// TIA Portal V19 export
FUNCTION_BLOCK "F_TwoHands_FB"   // FB93, F_LAD
TITLE = SAFE BUTTONS - TWO HANDS / ENABLING SWITCH / DEAD-MAN
// stored: Access Published
   VAR
      LB101 : "TwoHand_FB";
      LB111 : "TwoHand_FB";
      LB112 : "TwoHand_FB";
      LB113 : "TwoHand_FB";
      LB113_Welder : "TwoHand_FB";
      LB114_FeedA01 : "TwoHand_FB";
      LB114_FeedA02 : "TwoHand_FB";
      LB131 : "TwoHand_FB";
      LB131_FeedA01 : "TwoHand_FB";
      LB211 : "TwoHand_FB";
      LB212_FlyC : "TwoHand_FB";
      LB212_FeedA03 : "TwoHand_FB";
      LB311 : "TwoHand_FB";
   END_VAR
BEGIN

REGION Network 1: <<<< AREA 01 >>>
END_REGION

REGION Network 2: LB101 Two hands @ Zone 01 (Front of decoiler in load) / LB1.1 Two hands @ Area 01 Zone 01 (Front of decoiler in load)
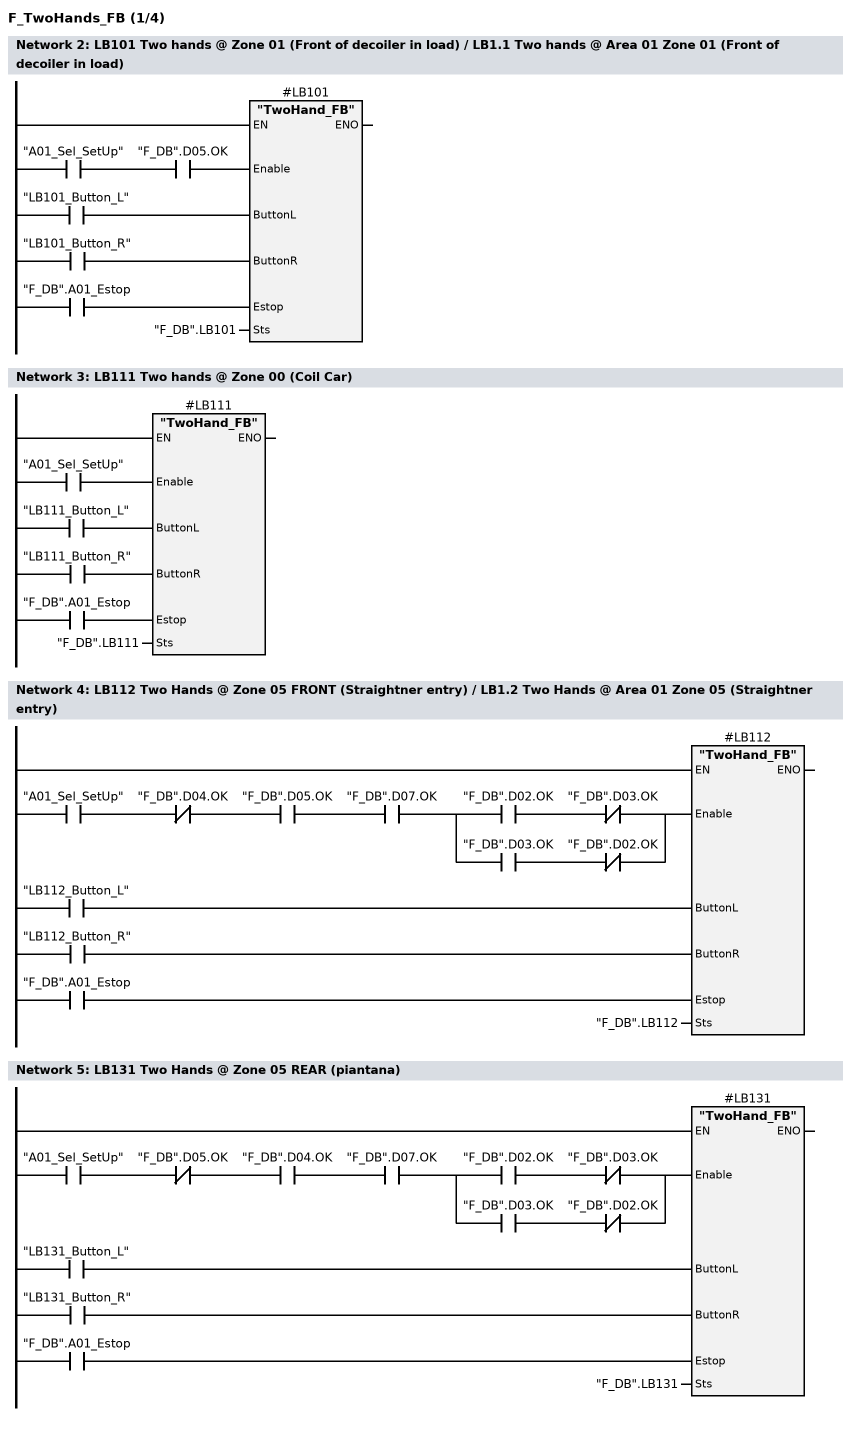
   RUNG wire#powerrail
      #LB101(Enable := wire#w1, ButtonL := wire#w2, ButtonR := wire#w3, Estop := wire#w4, Sts := "F_DB".LB101)
   END_RUNG
   RUNG wire#powerrail
      Contact( "A01_Sel_SetUp" )
      Contact( "F_DB".D05.OK )
   END_RUNG wire#w1
   RUNG wire#powerrail
      Contact( "LB101_Button_L" )
   END_RUNG wire#w2
   RUNG wire#powerrail
      Contact( "LB101_Button_R" )
   END_RUNG wire#w3
   RUNG wire#powerrail
      Contact( "F_DB".A01_Estop )
   END_RUNG wire#w4
   // the same network as SCL:
   #LB101(Enable := "A01_Sel_SetUp" AND "F_DB".D05.OK,   // "TwoHand_FB"
          ButtonL := "LB101_Button_L",
          ButtonR := "LB101_Button_R",
          Estop := "F_DB".A01_Estop,
          Sts := "F_DB".LB101);
END_REGION

REGION Network 3: LB111 Two hands @ Zone 00 (Coil Car)
   RUNG wire#powerrail
      #LB111(Enable := wire#w1, ButtonL := wire#w2, ButtonR := wire#w3, Estop := wire#w4, Sts := "F_DB".LB111)
   END_RUNG
   RUNG wire#powerrail
      Contact( "A01_Sel_SetUp" )
   END_RUNG wire#w1
   RUNG wire#powerrail
      Contact( "LB111_Button_L" )
   END_RUNG wire#w2
   RUNG wire#powerrail
      Contact( "LB111_Button_R" )
   END_RUNG wire#w3
   RUNG wire#powerrail
      Contact( "F_DB".A01_Estop )
   END_RUNG wire#w4
   // the same network as SCL:
   #LB111(Enable := "A01_Sel_SetUp",   // "TwoHand_FB"
          ButtonL := "LB111_Button_L",
          ButtonR := "LB111_Button_R",
          Estop := "F_DB".A01_Estop,
          Sts := "F_DB".LB111);
END_REGION

REGION Network 4: LB112 Two Hands @ Zone 05 FRONT (Straightner entry) / LB1.2 Two Hands @ Area 01 Zone 05 (Straightner entry)
   RUNG wire#powerrail
      #LB112(Enable := wire#w2, ButtonL := wire#w3, ButtonR := wire#w4, Estop := wire#w5, Sts := "F_DB".LB112)
   END_RUNG
   RUNG wire#powerrail
      Contact( "A01_Sel_SetUp" )
      I_Contact( "F_DB".D04.OK )
      Contact( "F_DB".D05.OK )
      Contact( "F_DB".D07.OK )
      wire#w1
      Contact( "F_DB".D02.OK )
      I_Contact( "F_DB".D03.OK )
   END_RUNG wire#w2
   RUNG wire#w1
      Contact( "F_DB".D03.OK )
      I_Contact( "F_DB".D02.OK )
   END_RUNG wire#w2
   RUNG wire#powerrail
      Contact( "LB112_Button_L" )
   END_RUNG wire#w3
   RUNG wire#powerrail
      Contact( "LB112_Button_R" )
   END_RUNG wire#w4
   RUNG wire#powerrail
      Contact( "F_DB".A01_Estop )
   END_RUNG wire#w5
   // the same network as SCL:
   #LB112(Enable := "A01_Sel_SetUp" AND NOT "F_DB".D04.OK AND "F_DB".D05.OK AND "F_DB".D07.OK AND (("F_DB".D02.OK AND NOT "F_DB".D03.OK) OR ("F_DB".D03.OK AND NOT "F_DB".D02.OK)),   // "TwoHand_FB"
          ButtonL := "LB112_Button_L",
          ButtonR := "LB112_Button_R",
          Estop := "F_DB".A01_Estop,
          Sts := "F_DB".LB112);
END_REGION

REGION Network 5: LB131 Two Hands @ Zone 05 REAR (piantana)
   RUNG wire#powerrail
      #LB131(Enable := wire#w2, ButtonL := wire#w3, ButtonR := wire#w4, Estop := wire#w5, Sts := "F_DB".LB131)
   END_RUNG
   RUNG wire#powerrail
      Contact( "A01_Sel_SetUp" )
      I_Contact( "F_DB".D05.OK )
      Contact( "F_DB".D04.OK )
      Contact( "F_DB".D07.OK )
      wire#w1
      Contact( "F_DB".D02.OK )
      I_Contact( "F_DB".D03.OK )
   END_RUNG wire#w2
   RUNG wire#w1
      Contact( "F_DB".D03.OK )
      I_Contact( "F_DB".D02.OK )
   END_RUNG wire#w2
   RUNG wire#powerrail
      Contact( "LB131_Button_L" )
   END_RUNG wire#w3
   RUNG wire#powerrail
      Contact( "LB131_Button_R" )
   END_RUNG wire#w4
   RUNG wire#powerrail
      Contact( "F_DB".A01_Estop )
   END_RUNG wire#w5
   // the same network as SCL:
   #LB131(Enable := "A01_Sel_SetUp" AND NOT "F_DB".D05.OK AND "F_DB".D04.OK AND "F_DB".D07.OK AND (("F_DB".D02.OK AND NOT "F_DB".D03.OK) OR ("F_DB".D03.OK AND NOT "F_DB".D02.OK)),   // "TwoHand_FB"
          ButtonL := "LB131_Button_L",
          ButtonR := "LB131_Button_R",
          Estop := "F_DB".A01_Estop,
          Sts := "F_DB".LB131);
END_REGION

REGION Network 6: LB113 Two Hands @ Zone 05 FRONT (Junction bench) / LB1.3 Two Hands @ Area 01 Zone 07 (Junction bench)
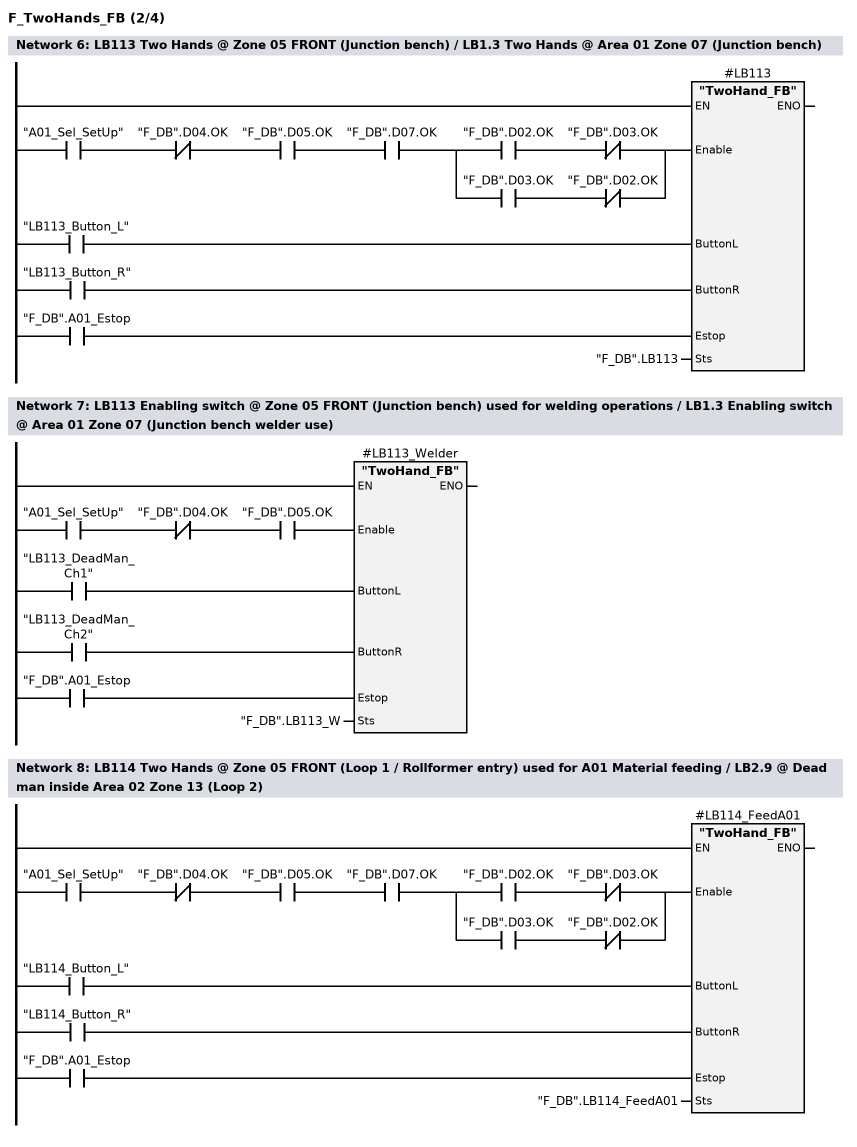
   RUNG wire#powerrail
      #LB113(Enable := wire#w2, ButtonL := wire#w3, ButtonR := wire#w4, Estop := wire#w5, Sts := "F_DB".LB113)
   END_RUNG
   RUNG wire#powerrail
      Contact( "A01_Sel_SetUp" )
      I_Contact( "F_DB".D04.OK )
      Contact( "F_DB".D05.OK )
      Contact( "F_DB".D07.OK )
      wire#w1
      Contact( "F_DB".D02.OK )
      I_Contact( "F_DB".D03.OK )
   END_RUNG wire#w2
   RUNG wire#w1
      Contact( "F_DB".D03.OK )
      I_Contact( "F_DB".D02.OK )
   END_RUNG wire#w2
   RUNG wire#powerrail
      Contact( "LB113_Button_L" )
   END_RUNG wire#w3
   RUNG wire#powerrail
      Contact( "LB113_Button_R" )
   END_RUNG wire#w4
   RUNG wire#powerrail
      Contact( "F_DB".A01_Estop )
   END_RUNG wire#w5
   // the same network as SCL:
   #LB113(Enable := "A01_Sel_SetUp" AND NOT "F_DB".D04.OK AND "F_DB".D05.OK AND "F_DB".D07.OK AND (("F_DB".D02.OK AND NOT "F_DB".D03.OK) OR ("F_DB".D03.OK AND NOT "F_DB".D02.OK)),   // "TwoHand_FB"
          ButtonL := "LB113_Button_L",
          ButtonR := "LB113_Button_R",
          Estop := "F_DB".A01_Estop,
          Sts := "F_DB".LB113);
END_REGION

REGION Network 7: LB113 Enabling switch @ Zone 05 FRONT (Junction bench) used for welding operations / LB1.3 Enabling switch @ Area 01 Zone 07 (Junction bench welder use)
   RUNG wire#powerrail
      #LB113_Welder(Enable := wire#w1, ButtonL := wire#w2, ButtonR := wire#w3, Estop := wire#w4, Sts := "F_DB".LB113_W)
   END_RUNG
   RUNG wire#powerrail
      Contact( "A01_Sel_SetUp" )
      I_Contact( "F_DB".D04.OK )
      Contact( "F_DB".D05.OK )
   END_RUNG wire#w1
   RUNG wire#powerrail
      Contact( "LB113_DeadMan_Ch1" )
   END_RUNG wire#w2
   RUNG wire#powerrail
      Contact( "LB113_DeadMan_Ch2" )
   END_RUNG wire#w3
   RUNG wire#powerrail
      Contact( "F_DB".A01_Estop )
   END_RUNG wire#w4
   // the same network as SCL:
   #LB113_Welder(Enable := "A01_Sel_SetUp" AND NOT "F_DB".D04.OK AND "F_DB".D05.OK,   // "TwoHand_FB"
                 ButtonL := "LB113_DeadMan_Ch1",
                 ButtonR := "LB113_DeadMan_Ch2",
                 Estop := "F_DB".A01_Estop,
                 Sts := "F_DB".LB113_W);
END_REGION

REGION Network 8: LB114 Two Hands @ Zone 05 FRONT (Loop 1 / Rollformer entry) used for A01 Material feeding / LB2.9 @ Dead man inside Area 02 Zone 13 (Loop 2)
   RUNG wire#powerrail
      #LB114_FeedA01(Enable := wire#w2, ButtonL := wire#w3, ButtonR := wire#w4, Estop := wire#w5, Sts := "F_DB".LB114_FeedA01)
   END_RUNG
   RUNG wire#powerrail
      Contact( "A01_Sel_SetUp" )
      I_Contact( "F_DB".D04.OK )
      Contact( "F_DB".D05.OK )
      Contact( "F_DB".D07.OK )
      wire#w1
      Contact( "F_DB".D02.OK )
      I_Contact( "F_DB".D03.OK )
   END_RUNG wire#w2
   RUNG wire#w1
      Contact( "F_DB".D03.OK )
      I_Contact( "F_DB".D02.OK )
   END_RUNG wire#w2
   RUNG wire#powerrail
      Contact( "LB114_Button_L" )
   END_RUNG wire#w3
   RUNG wire#powerrail
      Contact( "LB114_Button_R" )
   END_RUNG wire#w4
   RUNG wire#powerrail
      Contact( "F_DB".A01_Estop )
   END_RUNG wire#w5
   // the same network as SCL:
   #LB114_FeedA01(Enable := "A01_Sel_SetUp" AND NOT "F_DB".D04.OK AND "F_DB".D05.OK AND "F_DB".D07.OK AND (("F_DB".D02.OK AND NOT "F_DB".D03.OK) OR ("F_DB".D03.OK AND NOT "F_DB".D02.OK)),   // "TwoHand_FB"
                  ButtonL := "LB114_Button_L",
                  ButtonR := "LB114_Button_R",
                  Estop := "F_DB".A01_Estop,
                  Sts := "F_DB".LB114_FeedA01);
END_REGION

REGION Network 10: <<<< AREA 02 >>>
END_REGION

REGION Network 11: LB114 Two Hands @ Zone xx (Loop 1 / Rollformer entry) used for A02 material feeding
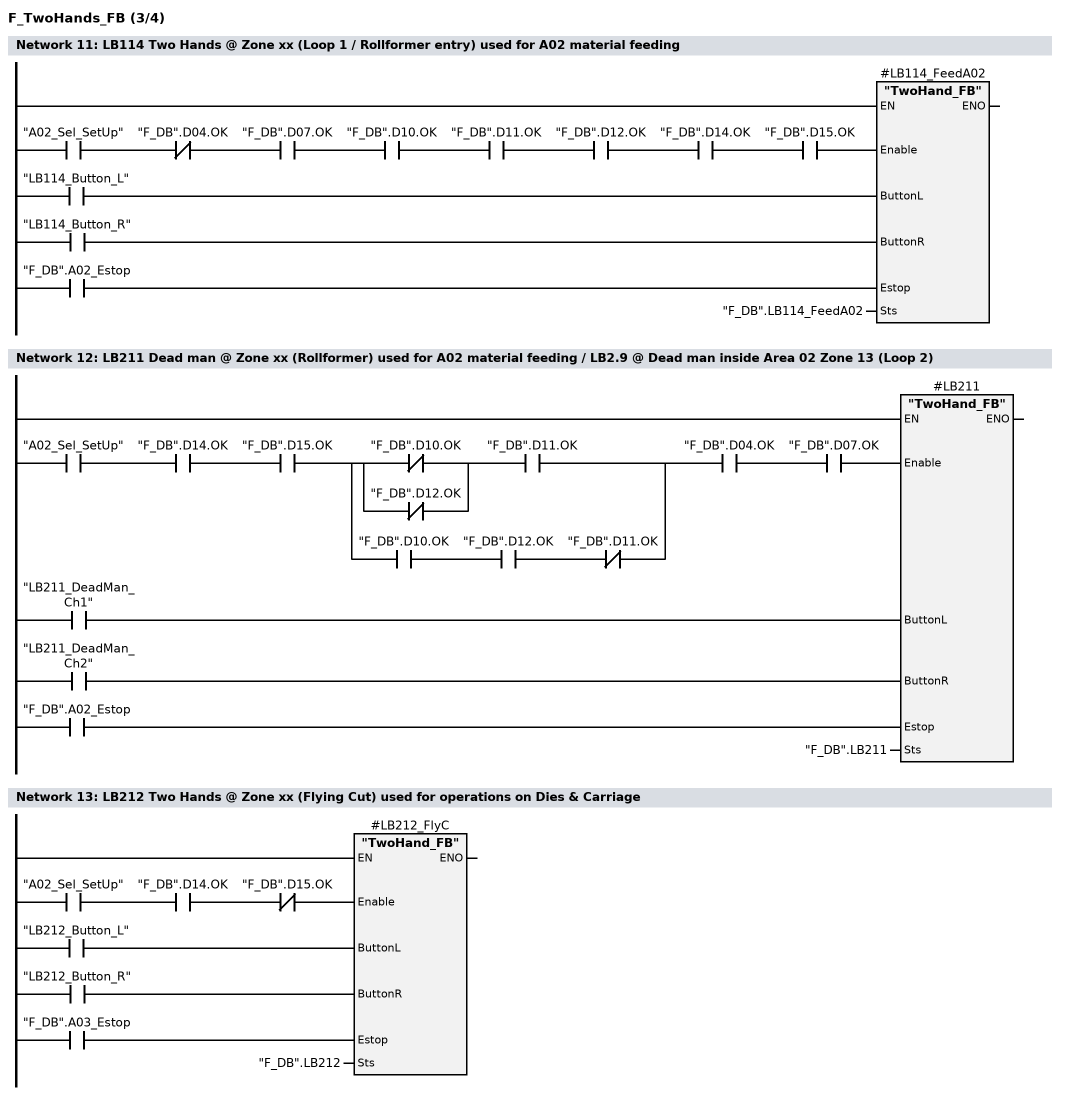
   RUNG wire#powerrail
      #LB114_FeedA02(Enable := wire#w1, ButtonL := wire#w2, ButtonR := wire#w3, Estop := wire#w4, Sts := "F_DB".LB114_FeedA02)
   END_RUNG
   RUNG wire#powerrail
      Contact( "A02_Sel_SetUp" )
      I_Contact( "F_DB".D04.OK )
      Contact( "F_DB".D07.OK )
      Contact( "F_DB".D10.OK )
      Contact( "F_DB".D11.OK )
      Contact( "F_DB".D12.OK )
      Contact( "F_DB".D14.OK )
      Contact( "F_DB".D15.OK )
   END_RUNG wire#w1
   RUNG wire#powerrail
      Contact( "LB114_Button_L" )
   END_RUNG wire#w2
   RUNG wire#powerrail
      Contact( "LB114_Button_R" )
   END_RUNG wire#w3
   RUNG wire#powerrail
      Contact( "F_DB".A02_Estop )
   END_RUNG wire#w4
   // the same network as SCL:
   #LB114_FeedA02(Enable := "A02_Sel_SetUp" AND NOT "F_DB".D04.OK AND "F_DB".D07.OK AND "F_DB".D10.OK AND "F_DB".D11.OK AND "F_DB".D12.OK AND "F_DB".D14.OK AND "F_DB".D15.OK,   // "TwoHand_FB"
                  ButtonL := "LB114_Button_L",
                  ButtonR := "LB114_Button_R",
                  Estop := "F_DB".A02_Estop,
                  Sts := "F_DB".LB114_FeedA02);
END_REGION

REGION Network 12: LB211 Dead man @ Zone xx (Rollformer) used for A02 material feeding / LB2.9 @ Dead man inside Area 02 Zone 13 (Loop 2)
   RUNG wire#powerrail
      #LB211(Enable := wire#w4, ButtonL := wire#w5, ButtonR := wire#w6, Estop := wire#w7, Sts := "F_DB".LB211)
   END_RUNG
   RUNG wire#powerrail
      Contact( "A02_Sel_SetUp" )
      Contact( "F_DB".D14.OK )
      Contact( "F_DB".D15.OK )
      wire#w1
      I_Contact( "F_DB".D10.OK )
      wire#w2
      Contact( "F_DB".D11.OK )
      wire#w3
      Contact( "F_DB".D04.OK )
      Contact( "F_DB".D07.OK )
   END_RUNG wire#w4
   RUNG wire#w1
      I_Contact( "F_DB".D12.OK )
   END_RUNG wire#w2
   RUNG wire#w1
      Contact( "F_DB".D10.OK )
      Contact( "F_DB".D12.OK )
      I_Contact( "F_DB".D11.OK )
   END_RUNG wire#w3
   RUNG wire#powerrail
      Contact( "LB211_DeadMan_Ch1" )
   END_RUNG wire#w5
   RUNG wire#powerrail
      Contact( "LB211_DeadMan_Ch2" )
   END_RUNG wire#w6
   RUNG wire#powerrail
      Contact( "F_DB".A02_Estop )
   END_RUNG wire#w7
   // the same network as SCL:
   #LB211(Enable := "A02_Sel_SetUp" AND "F_DB".D14.OK AND "F_DB".D15.OK AND (((NOT "F_DB".D10.OK OR NOT "F_DB".D12.OK) AND "F_DB".D11.OK) OR ("F_DB".D10.OK AND "F_DB".D12.OK AND NOT "F_DB".D11.OK)) AND "F_DB".D04.OK AND "F_DB".D07.OK,   // "TwoHand_FB"
          ButtonL := "LB211_DeadMan_Ch1",
          ButtonR := "LB211_DeadMan_Ch2",
          Estop := "F_DB".A02_Estop,
          Sts := "F_DB".LB211);
END_REGION

REGION Network 13: LB212 Two Hands @ Zone xx (Flying Cut) used for operations on Dies & Carriage
   RUNG wire#powerrail
      #LB212_FlyC(Enable := wire#w1, ButtonL := wire#w2, ButtonR := wire#w3, Estop := wire#w4, Sts := "F_DB".LB212)
   END_RUNG
   RUNG wire#powerrail
      Contact( "A02_Sel_SetUp" )
      Contact( "F_DB".D14.OK )
      I_Contact( "F_DB".D15.OK )
   END_RUNG wire#w1
   RUNG wire#powerrail
      Contact( "LB212_Button_L" )
   END_RUNG wire#w2
   RUNG wire#powerrail
      Contact( "LB212_Button_R" )
   END_RUNG wire#w3
   RUNG wire#powerrail
      Contact( "F_DB".A03_Estop )
   END_RUNG wire#w4
   // the same network as SCL:
   #LB212_FlyC(Enable := "A02_Sel_SetUp" AND "F_DB".D14.OK AND NOT "F_DB".D15.OK,   // "TwoHand_FB"
               ButtonL := "LB212_Button_L",
               ButtonR := "LB212_Button_R",
               Estop := "F_DB".A03_Estop,
               Sts := "F_DB".LB212);
END_REGION

REGION Network 14: LB212 Two Hands @ Zone xx (Flying Cut) used for A02 material feeding
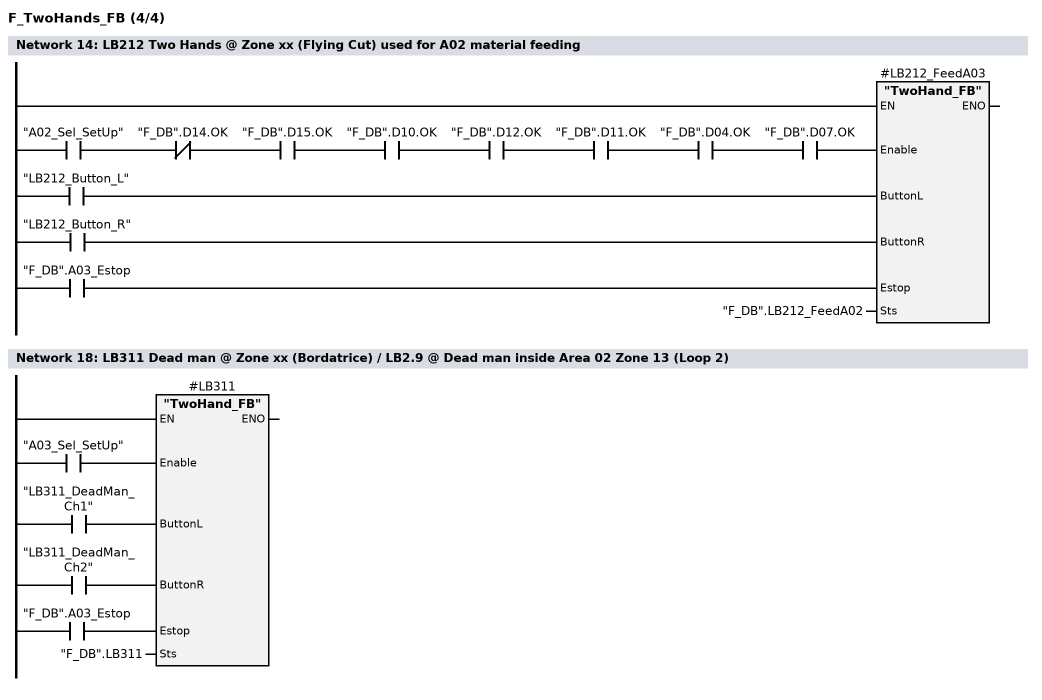
   RUNG wire#powerrail
      #LB212_FeedA03(Enable := wire#w1, ButtonL := wire#w2, ButtonR := wire#w3, Estop := wire#w4, Sts := "F_DB".LB212_FeedA02)
   END_RUNG
   RUNG wire#powerrail
      Contact( "A02_Sel_SetUp" )
      I_Contact( "F_DB".D14.OK )
      Contact( "F_DB".D15.OK )
      Contact( "F_DB".D10.OK )
      Contact( "F_DB".D12.OK )
      Contact( "F_DB".D11.OK )
      Contact( "F_DB".D04.OK )
      Contact( "F_DB".D07.OK )
   END_RUNG wire#w1
   RUNG wire#powerrail
      Contact( "LB212_Button_L" )
   END_RUNG wire#w2
   RUNG wire#powerrail
      Contact( "LB212_Button_R" )
   END_RUNG wire#w3
   RUNG wire#powerrail
      Contact( "F_DB".A03_Estop )
   END_RUNG wire#w4
   // the same network as SCL:
   #LB212_FeedA03(Enable := "A02_Sel_SetUp" AND NOT "F_DB".D14.OK AND "F_DB".D15.OK AND "F_DB".D10.OK AND "F_DB".D12.OK AND "F_DB".D11.OK AND "F_DB".D04.OK AND "F_DB".D07.OK,   // "TwoHand_FB"
                  ButtonL := "LB212_Button_L",
                  ButtonR := "LB212_Button_R",
                  Estop := "F_DB".A03_Estop,
                  Sts := "F_DB".LB212_FeedA02);
END_REGION

REGION Network 17: <<<< AREA 03 >>>
END_REGION

REGION Network 18: LB311 Dead man @ Zone xx (Bordatrice) / LB2.9 @ Dead man inside Area 02 Zone 13 (Loop 2)
   RUNG wire#powerrail
      #LB311(Enable := wire#w1, ButtonL := wire#w2, ButtonR := wire#w3, Estop := wire#w4, Sts := "F_DB".LB311)
   END_RUNG
   RUNG wire#powerrail
      Contact( "A03_Sel_SetUp" )
   END_RUNG wire#w1
   RUNG wire#powerrail
      Contact( "LB311_DeadMan_Ch1" )
   END_RUNG wire#w2
   RUNG wire#powerrail
      Contact( "LB311_DeadMan_Ch2" )
   END_RUNG wire#w3
   RUNG wire#powerrail
      Contact( "F_DB".A03_Estop )
   END_RUNG wire#w4
   // the same network as SCL:
   #LB311(Enable := "A03_Sel_SetUp",   // "TwoHand_FB"
          ButtonL := "LB311_DeadMan_Ch1",
          ButtonR := "LB311_DeadMan_Ch2",
          Estop := "F_DB".A03_Estop,
          Sts := "F_DB".LB311);
END_REGION
END_FUNCTION_BLOCK
